ABB RobotStudio station: ___new.rsstn

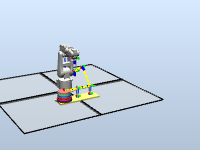
Station 叠放盘子_1 (saved by RobotStudio 6.8.8148.134)
Controller System36
  mechanical unit ROB_1: IRB120_3_58__01, 6 joints, base frame (0, 0, 0) mm
Layout (positions relative to the parent item):
  - IRB120_3_58__01 [mechanism, from Robots\IRB120_3_58_G_01.rslib] at (0, 0, 0) mm; joint values [0, 0, 0, 0, 1.5708, 0] (rad or m)
  - 放置架 [part] at (381.81, -51.15, -51.29) mm, rotated rx 90 ry 0 rz 90 deg
  - 物料170 [part]
  - 物料175 [part]
  - 物料180 [part]
  - 物料185 [part]
  - 物料190 [part]
  - 物料195 [part]
  - 物料200 [part]
  - 物料205 [part]
  - 物料210 [part]
  - SC_Sukcer [smart component] at (0, 0, 0) mm
      signals: DI di01_Sucker
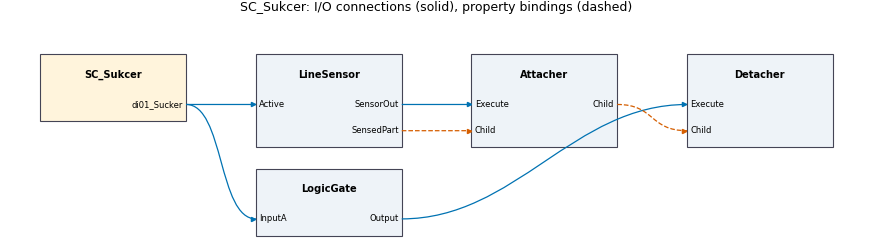
      connections:
        SC_Sukcer.di01_Sucker -> LineSensor.Active
        LogicGate.Output -> Detacher.Execute
        LineSensor.SensorOut -> Attacher.Execute
        SC_Sukcer.di01_Sucker -> LogicGate.InputA
        LineSensor.SensedPart => Attacher.Child
        Attacher.Child => Detacher.Child
    - LineSensor [smart component, from Components\LineSensor.rslib]
        properties: Start=[0.302 -0.025 0.3802]; End=[0.302 -0.025 0.3912]; Radius=0.005; SensedPart=(none); SensedPoint=[0 0 0]
      - _sensorPart_ [part]
    - Attacher [smart component, from Components\Attacher.rslib]
        properties: Parent=SC_Sukcer; Flange=0; Child=(none); Mount=false; Offset=[0 0 0]; Orientation=[0 0 0]
    - Detacher [smart component, from Components\Detacher.rslib]
        properties: Child=(none); KeepPosition=true
    - LogicGate [smart component, from Components\LogicGate.rslib]
        properties: Operator=NOT; Delay=0
    - sucker [mechanism] at (302, 0, 558) mm, rotated rx 180 ry 0 rz 180 deg
        TCP sucker at (0, 0, 166.6) mm
        links: 吸盘
  - 组_2 [graphiccomponentgroup] at (0, 0, 174.72) mm, rotated rx 180 ry 0 rz 0 deg
    - 组_3 [graphiccomponentgroup]
    - 物料180_2 [part]
    - 物料185_2 [part]
    - 物料190_2 [part]
    - 物料195_2 [part]
    - 物料200_2 [part]
    - 物料205_2 [part]
    - 物料210_2 [part]
    - 物料175_2 [part]
    - 物料170_2 [part]
  - 组_4 [graphiccomponentgroup] at (0, 200, 1.02) mm
    - 物料170_3 [part]
    - 物料175_3 [part]
    - 物料180_3 [part]
    - 物料190_3 [part]
    - 物料185_3 [part]
    - 物料195_3 [part]
    - 物料200_3 [part]
    - 物料205_3 [part]
    - 物料210_3 [part]
  - 框架_1 [frame] at (0, 0, 172.2) mm
Attachment: sucker is attached to IRB120_3_58__01 / Link6
Attachment: SC_Sukcer is attached to IRB120_3_58__01 / Link6
EventTableEntry 1488: Group=, Trigger=dosucker0 1489, Actions=[EventTableActionAttach 1490], Comment=, ActivationMode=2, Cyclic=false
EventTableTriggerIO 1489: IOValue=[1], IRC5Controller=? -1, Operator=0, SignalSource=? -1
EventTableActionAttach 1490: AttachmentParent=sucker 1484, AttachmentChild=物料170 1463, MountObject=false, Offset=[X=1, Y=0, Z=0, W=0, X=0, Y=1, Z=0, W=0, X=0, Y=0, Z=1, W=0, X=0, Y=0, Z=0, W=1], FlangeIndext=0, FindNearest=false
EventTableEntry 1491: Group=, Trigger=dosucker0 1492, Actions=[EventTableActionDetach 1493], Comment=, ActivationMode=2, Cyclic=false
EventTableTriggerIO 1492: IOValue=[0], IRC5Controller=? -1, Operator=0, SignalSource=? -1
EventTableActionDetach 1493: AttachmentParent=sucker 1484, AttachmentChild=物料170 1463
EventTableTriggerIO 1630: IOValue=[1], IRC5Controller=? -1, Operator=0, SignalSource=? -1
EventTableTriggerIO 1631: IOValue=[1], IRC5Controller=? -1, Operator=0, SignalSource=? -1
EventTableTriggerIO 1632: IOValue=[1], IRC5Controller=? -1, Operator=0, SignalSource=? -1
EventTableTriggerIO 1633: IOValue=[1], IRC5Controller=? -1, Operator=0, SignalSource=? -1
EventTableTriggerIO 1634: IOValue=[1], IRC5Controller=? -1, Operator=0, SignalSource=? -1
EventTableTriggerIO 1635: IOValue=[1], IRC5Controller=? -1, Operator=0, SignalSource=? -1
EventTableTriggerIO 1636: IOValue=[1], IRC5Controller=? -1, Operator=0, SignalSource=? -1
EventTableTriggerIO 1637: IOValue=[1], IRC5Controller=? -1, Operator=0, SignalSource=? -1
EventTableTriggerIO 1638: IOValue=[1], IRC5Controller=? -1, Operator=0, SignalSource=? -1
EventTableTriggerIO 1639: IOValue=[1], IRC5Controller=? -1, Operator=0, SignalSource=? -1
EventTableTriggerIO 1640: IOValue=[1], IRC5Controller=? -1, Operator=0, SignalSource=? -1
EventTableTriggerIO 1641: IOValue=[0], IRC5Controller=? -1, Operator=0, SignalSource=? -1
EventTableTriggerIO 1642: IOValue=[0], IRC5Controller=? -1, Operator=0, SignalSource=? -1
EventTableTriggerIO 1643: IOValue=[0], IRC5Controller=? -1, Operator=0, SignalSource=? -1
EventTableTriggerIO 1644: IOValue=[0], IRC5Controller=? -1, Operator=0, SignalSource=? -1
EventTableTriggerIO 1645: IOValue=[0], IRC5Controller=? -1, Operator=0, SignalSource=? -1
EventTableTriggerIO 1646: IOValue=[0], IRC5Controller=? -1, Operator=0, SignalSource=? -1
EventTableTriggerIO 1647: IOValue=[0], IRC5Controller=? -1, Operator=0, SignalSource=? -1
EventTableTriggerIO 1648: IOValue=[0], IRC5Controller=? -1, Operator=0, SignalSource=? -1
EventTableTriggerIO 1649: IOValue=[0], IRC5Controller=? -1, Operator=0, SignalSource=? -1
EventTableTriggerIO 1650: IOValue=[0], IRC5Controller=? -1, Operator=0, SignalSource=? -1
EventTableTriggerIO 1651: IOValue=[0], IRC5Controller=? -1, Operator=0, SignalSource=? -1
EventTableTriggerIO 2136: IOValue=[1], IRC5Controller=? -1, Operator=0, SignalSource=? -1
EventTableTriggerIO 2137: IOValue=[1], IRC5Controller=? -1, Operator=0, SignalSource=? -1
EventTableTriggerIO 2138: IOValue=[1], IRC5Controller=? -1, Operator=0, SignalSource=? -1
EventTableTriggerIO 2139: IOValue=[1], IRC5Controller=? -1, Operator=0, SignalSource=? -1
EventTableTriggerIO 2140: IOValue=[1], IRC5Controller=? -1, Operator=0, SignalSource=? -1
EventTableTriggerIO 2141: IOValue=[0], IRC5Controller=? -1, Operator=0, SignalSource=? -1
EventTableTriggerIO 2142: IOValue=[0], IRC5Controller=? -1, Operator=0, SignalSource=? -1
EventTableTriggerIO 2143: IOValue=[0], IRC5Controller=? -1, Operator=0, SignalSource=? -1
EventTableTriggerIO 2144: IOValue=[0], IRC5Controller=? -1, Operator=0, SignalSource=? -1
EventTableTriggerIO 2145: IOValue=[0], IRC5Controller=? -1, Operator=0, SignalSource=? -1
Station logic (signal -> signal, property => property):
  System38.doSucker -> SC_Sukcer.di01_Sucker
  System36.doSucker -> SC_Sukcer.di01_Sucker
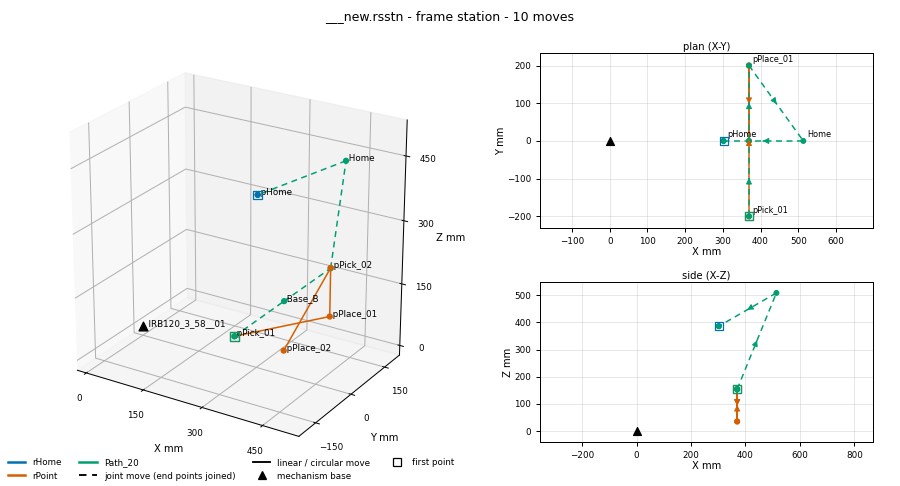
[picture p0: tool path of ___new.rsstn in frame station, 10 of 14 moves have a stored position in this frame; points joined in program order, loops and branches not executed]
Targets, tools, work objects and paths stored in the station, written as RAPID:
! task T_ROB1
MODULE CalibData
  PERS tooldata sucker:=[TRUE,[[0,0,172.2],[1,0,0,0]],[1,[0,-0.001,66.931],[1,0,0,0],0,0,0]];
  TASK PERS wobjdata Workobject_1:=[FALSE,TRUE,"",[[0,0,0],[1,0,0,0]],[[0,0,0],[1,0,0,0]]];
ENDMODULE

! task T_ROB1
MODULE Module1
  CONST robtarget pHome:=[[302,0,385.8],[0,0,1,0],[0,0,0,0],[9E+09,9E+09,9E+09,9E+09,9E+09,9E+09]];
  CONST robtarget pPick_01:=[[369.384508809,-200.000304101,154.139549259],[-0.000000029,0.000000006,1,0.000000025],[-1,0,-1,0],[9E+09,9E+09,9E+09,9E+09,9E+09,9E+09]];
  CONST robtarget rPlace_01:=[[369.384499755,199.9994975,35.576845668],[-0.000000023,0.000000004,1,0.000000028],[0,0,0,0],[9E+09,9E+09,9E+09,9E+09,9E+09,9E+09]];
  CONST robtarget rPick_02:=[[369.384502218,199.999498834,154.94336103],[-0.000000023,0.000000011,1,0.000000028],[0,0,0,0],[9E+09,9E+09,9E+09,9E+09,9E+09,9E+09]];
  CONST robtarget rPlace_02:=[[369.384497639,-0.000490748,35.795418953],[-0.000000022,0.000000011,1,0.000000028],[-1,0,-1,0],[9E+09,9E+09,9E+09,9E+09,9E+09,9E+09]];
  CONST robtarget pPlace_01:=[[369.384499755,199.9994975,35.576845668],[-0.000000023,0.000000004,1,0.000000028],[0,0,0,0],[9E+09,9E+09,9E+09,9E+09,9E+09,9E+09]];
  CONST robtarget pPick_02:=[[369.384502218,199.999498834,154.94336103],[-0.000000023,0.000000011,1,0.000000028],[0,0,0,0],[9E+09,9E+09,9E+09,9E+09,9E+09,9E+09]];
  CONST robtarget pPlace_02:=[[369.384497639,-0.000490748,35.795418953],[-0.000000022,0.000000011,1,0.000000028],[-1,0,-1,0],[9E+09,9E+09,9E+09,9E+09,9E+09,9E+09]];
  PROC rHome()
    MoveJ pHome,v4000,fine,sucker\WObj:=wobj0;
  ENDPROC
  PROC rPoint()
    MoveL pPick_01,v4000,z100,sucker\WObj:=Workobject_1;
    MoveL pPlace_01,v4000,z100,sucker\WObj:=Workobject_1;
    MoveL pPick_02,v4000,z100,sucker\WObj:=Workobject_1;
    MoveL pPlace_02,v4000,z100,sucker\WObj:=Workobject_1;
  ENDPROC
  PROC main()
    rInitall;
    rPick_01;
    rHome;
  ENDPROC
  PROC rPick_01()
    MoveL Offs(pPick_01,0,0,zPick_01+200),v4000,z100,sucker\WObj:=Workobject_1;
    MoveL Offs(pPick_01,0,0,zPick_01+50),v4000,z100,sucker\WObj:=Workobject_1;
    MoveL Offs(pPick_01,0,0,zPick_01),v4000,fine,sucker\WObj:=Workobject_1;
    Set doSucker;
    WaitTime 0.5;
    MoveL Offs(pPick_01,0,0,zPick_01+200),v4000,z100,sucker\WObj:=Workobject_1;
  ENDPROC
  PROC rInitall()
    rHome;
  ENDPROC
ENDMODULE

! task T_ROB1
MODULE CalibData
  PERS tooldata sucker:=[TRUE,[[0,0,172.2],[1,0,0,0]],[1,[0,-0.001,66.931],[1,0,0,0],0,0,0]];
ENDMODULE

! task T_ROB1
MODULE Module1
  CONST robtarget Home:=[[513.483403604,0,507.9],[0.5,0,0.866025404,0],[0,0,0,0],[9E+09,9E+09,9E+09,9E+09,9E+09,9E+09]];
  CONST robtarget Setout:=[[302,0,385.8],[0,0,1,0],[0,0,0,0],[9E+09,9E+09,9E+09,9E+09,9E+09,9E+09]];
  CONST robtarget Base_A:=[[369.385,-200,154.14],[0,0,1,0],[0,0,0,0],[9E+09,9E+09,9E+09,9E+09,9E+09,9E+09]];
  CONST robtarget Base_B:=[[369.385,0,154.14],[0,0,1,0],[0,0,0,0],[9E+09,9E+09,9E+09,9E+09,9E+09,9E+09]];
  CONST robtarget Base_C:=[[369.385,200,154.14],[0,0,1,0],[0,0,0,0],[9E+09,9E+09,9E+09,9E+09,9E+09,9E+09]];
  PROC Path_20()
    MoveJ Base_A,v1000,z100,sucker\WObj:=wobj0;
    MoveJ Base_B,v1000,z100,sucker\WObj:=wobj0;
    MoveJ Base_C,v1000,z100,sucker\WObj:=wobj0;
    MoveJ Home,v1000,z100,sucker\WObj:=wobj0;
    MoveJ Setout,v1000,z100,sucker\WObj:=wobj0;
  ENDPROC
ENDMODULE

